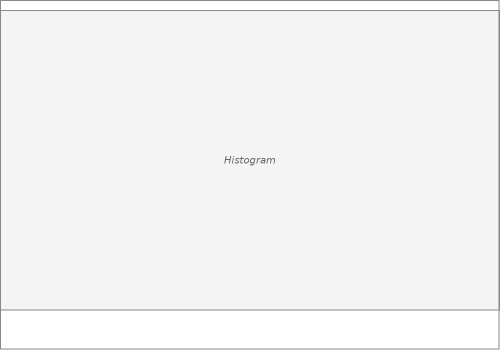
VISUALIZATION Frame_Trend_Einzel  // 500x350
VAR_IN_OUT
	itemValue : ARRAY[1..GVL_Const.gc_Max_ITEMS] OF REAL;
END_VAR
    Histogram (0,10 500x300), scale format: %.2f, scale -0.25..1.25
        p1518820177: itemValue
        p102497268: itemValue
        p788070771: ARRAY [1..GVL_Const.gc_Max_ITEMS] OF REAL
END_VISUALIZATION

(* stored: Version 1.1.0.1, ProductVersion 3.1.4020.12
   Visu Frame_Trend_Einzel: Id {380b1ef1-6b55-49c2-b7ec-bba4f9b81c7b} *)
